// TIA Portal V20 export
VAR_GLOBAL   // PLC tag table "ConvConstantC1"
END_VAR
VAR_GLOBAL CONSTANT   // user constants
   minC1 : Int := 3001;
   maxC1 : Int := 3054;
   "Conveyor_C1.1.1" : Int := 3001;
   "Conveyor_C1.1.2" : Int := 3002;
   "Conveyor_C1.1.3" : Int := 3003;
   "MABS_C1.2.1" : Int := 3051;
   "MABS_C1.2.2" : Int := 3052;
   "Conveyor_C1.9.1" : Int := 3031;
   "Conveyor_C1.10.1" : Int := 3032;
   "Conveyor_C1.11.1" : Int := 3033;
   "Conveyor_C1.11.2" : Int := 3034;
   "Conveyor_C1.12.1" : Int := 3035;
   "Conveyor_C1.12.2" : Int := 3036;
   "Conveyor_C1.12.3" : Int := 3037;
   "Transfer_C1.13.1" : Int := 3053;
   "Transfer_C1.14.1" : Int := 3054;
   "Conveyor_C1.15.2" : Int := 3038;
   "Conveyor_C1.15.3" : Int := 3039;
   "Conveyor_C1.15.4" : Int := 3040;
   "Conveyor_C1.16.1" : Int := 3041;
   "Conveyor_C1.18.1" : Int := 3042;
   "Conveyor_C1.18.2" : Int := 3043;
   "Conveyor_C1.18.3" : Int := 3044;
   "Conveyor_C1.18.4" : Int := 3045;
   "Conveyor_C1.18.5" : Int := 3046;
   "Conveyor_C1.18.6" : Int := 3047;
   "Conveyor_C1.18.7" : Int := 3048;
   "Conveyor_C1.19.1" : Int := 3049;
   "Conveyor_C1.20.2" : Int := 3050;
   "Conveyor_C1.3.1" : Int := 3004;
   "Conveyor_C1.3.2" : Int := 3005;
   "Conveyor_C1.3.3" : Int := 3006;
   "Conveyor_C1.3.4" : Int := 3007;
   "Conveyor_C1.3.5" : Int := 3008;
   "Conveyor_C1.3.6" : Int := 3009;
   "Conveyor_C1.3.7" : Int := 3010;
   "Conveyor_C1.3.8" : Int := 3011;
   "Conveyor_C1.3.9" : Int := 3012;
   "Conveyor_C1.3.10" : Int := 3013;
   "Conveyor_C1.4.1" : Int := 3014;
   "Conveyor_C1.4.2" : Int := 3015;
   "Conveyor_C1.4.3" : Int := 3016;
   "Conveyor_C1.4.4" : Int := 3017;
   "Conveyor_C1.5.1" : Int := 3018;
   "Conveyor_C1.6.1" : Int := 3019;
   "Conveyor_C1.6.2" : Int := 3020;
   "Conveyor_C1.7.1" : Int := 3021;
   "Conveyor_C1.7.2" : Int := 3022;
   "Conveyor_C1.7.3" : Int := 3023;
   "Conveyor_C1.7.4" : Int := 3024;
   "Conveyor_C1.7.5" : Int := 3025;
   "Conveyor_C1.7.6" : Int := 3026;
   "Conveyor_C1.7.7" : Int := 3027;
   "Conveyor_C1.7.8" : Int := 3028;
   "Conveyor_C1.7.9" : Int := 3029;
   "Conveyor_C1.7.10" : Int := 3030;
END_VAR
